FUNCTION_BLOCK FbStirControl IMPLEMENTS IStirControl

VAR_OUTPUT
	VFDSetpointOutput : LREAL;
END_VAR
VAR
END_VAR

{warning 'add property implementation'}
PROPERTY pSetpoint : LREAL
GET
pSetpoint := VFDSetpointOutput;
END_GET
END_PROPERTY

{warning 'add method implementation '}
METHOD StirControl : LREAL
VAR_INPUT
	i : INT;
END_VAR

IF IO.Reactors[i].VFD.bStart THEN
	VFDSetpointOutput := IO.Reactors[i].VFD.nRPMSetPointScaled;
ELSE
	VFDSetpointOutput := 0;		
END_IF
END_METHOD

END_FUNCTION_BLOCK

(* stored: Version 1.1.0.1, ProductVersion 3.1.4024.9
   POU FbStirControl: Id {c7a27a94-a89c-4e9d-b986-f8824acce40d}, SpecialFunc None
   Property pSetpoint: Id {8d188022-86b1-4051-9705-09833a301424}
   Get Get: Id {787095fb-b933-4ce0-8ba3-2c5a54cea94c}
   Method StirControl: Id {35bcf2e5-3ffe-4f7d-89ad-8ffc3320cb8d} *)
